% RSLogix 500 project P4_KOBIERSKI_M.RSS, saved by version 8.30.00.16 %
PROJECT "UNTITLED"    % processor: Bul.1763 MicroLogix 1100 Series B %

PROGRAM FILES
  LAD 2 "MAIN"  3 rungs
  LAD 3 "IO"  7 rungs
  LAD 4 "CYCLE"  11 rungs
  LAD 5 "STATES"  7 rungs

DATA FILES
  O0 OUTPUT  4 elements
  I1 INPUT  6 elements
  S2 STATUS  66 elements
  B3 BINARY  3 elements
  T4 TIMER  3 elements
  C5 COUNTER  1 elements
  R6 CONTROL  1 elements
  N7 INTEGER  2 elements
  F8 FLOAT  1 elements

LADDER 2 "MAIN"
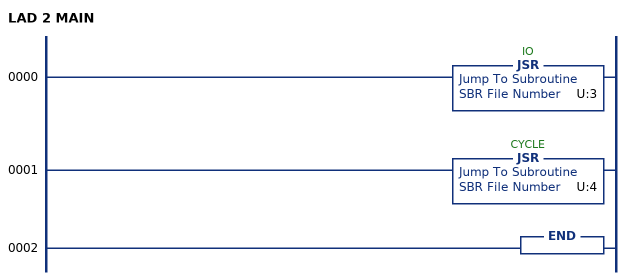
% Rung: 0 %
SOR JSR U:3 EOR
%   U:3  "IO" %
% Rung: 1 %
SOR JSR U:4 EOR
%   U:4  "CYCLE" %
% Rung: 2 %
SOR END EOR

LADDER 3 "IO"
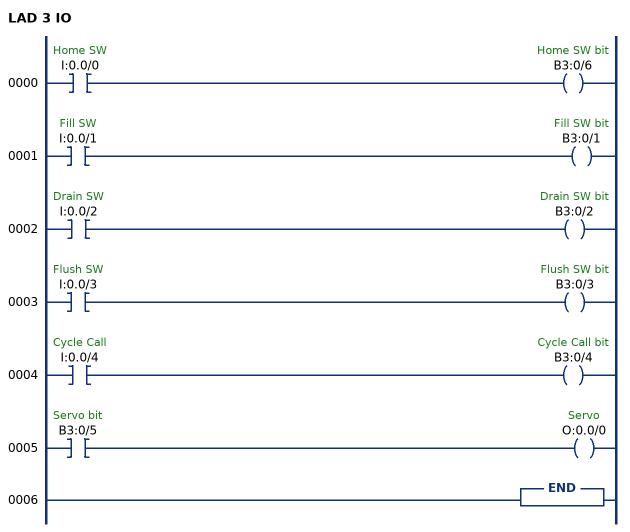
% Rung: 0 %
SOR XIC I:0.0/0 OTE B3:0/6 EOR
%   I:0.0/0  "Home SW" %
%   B3:0/6  "Home SW bit" %
% Rung: 1 %
SOR XIC I:0.0/1 OTE B3:0/1 EOR
%   I:0.0/1  "Fill SW" %
%   B3:0/1  "Fill SW bit" %
% Rung: 2 %
SOR XIC I:0.0/2 OTE B3:0/2 EOR
%   I:0.0/2  "Drain SW" %
%   B3:0/2  "Drain SW bit" %
% Rung: 3 %
SOR XIC I:0.0/3 OTE B3:0/3 EOR
%   I:0.0/3  "Flush SW" %
%   B3:0/3  "Flush SW bit" %
% Rung: 4 %
SOR XIC I:0.0/4 OTE B3:0/4 EOR
%   I:0.0/4  "Cycle Call" %
%   B3:0/4  "Cycle Call bit" %
% Rung: 5 %
SOR XIC B3:0/5 OTE O:0.0/0 EOR
%   B3:0/5  "Servo bit" %
%   O:0.0/0  "Servo" %
% Rung: 6 %
SOR END EOR

LADDER 4 "CYCLE"
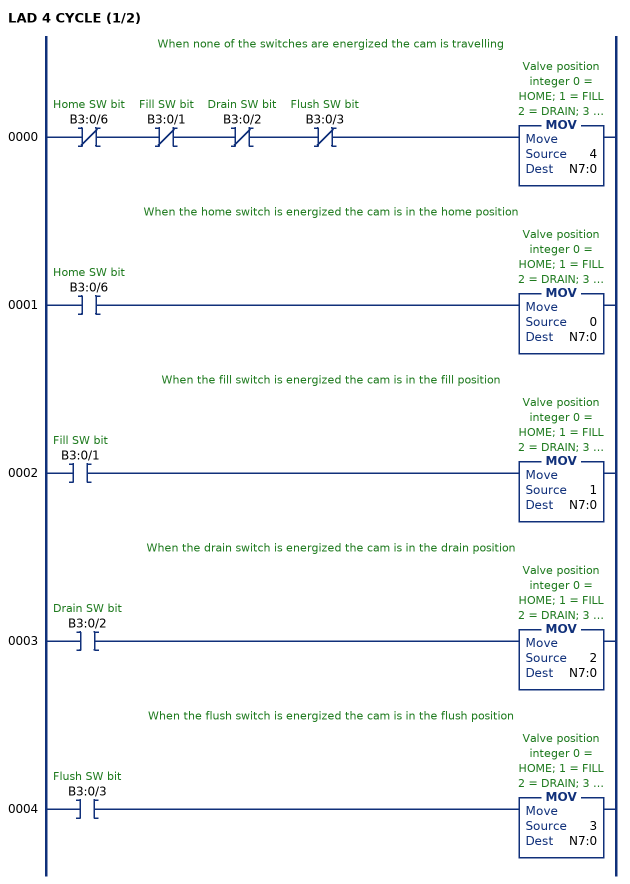
% Rung: 0 %
% When none of the switches are energized the cam is travelling %
SOR XIO B3:0/6 XIO B3:0/1 XIO B3:0/2 XIO B3:0/3 MOV 4 N7:0 EOR
%   B3:0/6  "Home SW bit" %
%   B3:0/1  "Fill SW bit" %
%   B3:0/2  "Drain SW bit" %
%   B3:0/3  "Flush SW bit" %
%   N7:0  "Valve position integer 0 = HOME; 1 = FILL 2 = DRAIN; 3 = FLUSH 4 = TRAVELLING" %
% Rung: 1 %
% When the home switch is energized the cam is in the home position %
SOR XIC B3:0/6 MOV 0 N7:0 EOR
%   B3:0/6  "Home SW bit" %
%   N7:0  "Valve position integer 0 = HOME; 1 = FILL 2 = DRAIN; 3 = FLUSH 4 = TRAVELLING" %
% Rung: 2 %
% When the fill switch is energized the cam is in the fill position %
SOR XIC B3:0/1 MOV 1 N7:0 EOR
%   B3:0/1  "Fill SW bit" %
%   N7:0  "Valve position integer 0 = HOME; 1 = FILL 2 = DRAIN; 3 = FLUSH 4 = TRAVELLING" %
% Rung: 3 %
% When the drain switch is energized the cam is in the drain position %
SOR XIC B3:0/2 MOV 2 N7:0 EOR
%   B3:0/2  "Drain SW bit" %
%   N7:0  "Valve position integer 0 = HOME; 1 = FILL 2 = DRAIN; 3 = FLUSH 4 = TRAVELLING" %
% Rung: 4 %
% When the flush switch is energized the cam is in the flush position %
SOR XIC B3:0/3 MOV 3 N7:0 EOR
%   B3:0/3  "Flush SW bit" %
%   N7:0  "Valve position integer 0 = HOME; 1 = FILL 2 = DRAIN; 3 = FLUSH 4 = TRAVELLING" %

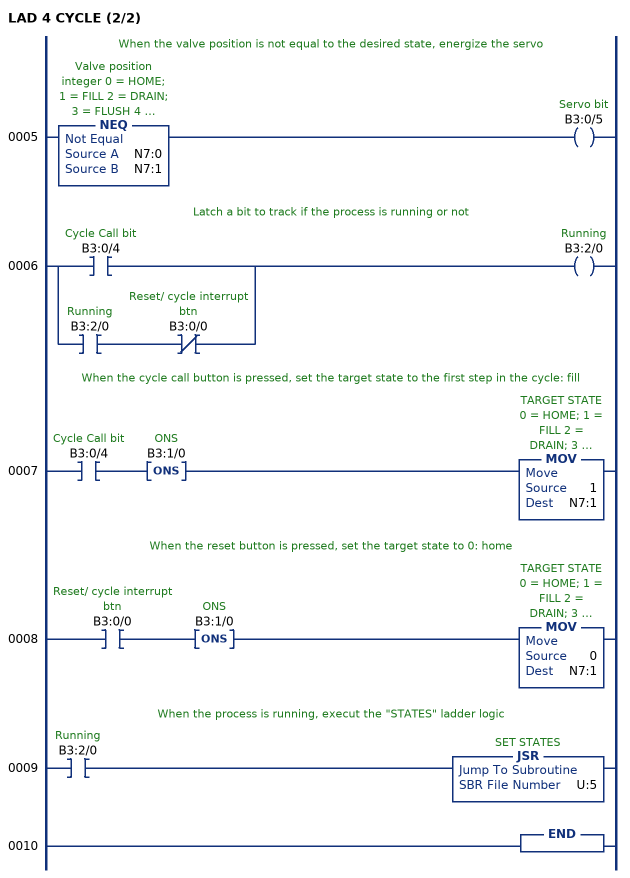
% Rung: 5 %
% When the valve position is not equal to the desired state, energize the servo %
SOR NEQ N7:0 N7:1 OTE B3:0/5 EOR
%   N7:0  "Valve position integer 0 = HOME; 1 = FILL 2 = DRAIN; 3 = FLUSH 4 = TRAVELLING" %
%   N7:1  "TARGET STATE 0 = HOME; 1 = FILL 2 = DRAIN; 3 = FLUSH" %
%   B3:0/5  "Servo bit" %
% Rung: 6 %
% Latch a bit to track if the process is running or not %
SOR BST XIC B3:0/4 NXB XIC B3:2/0 XIO B3:0/0 BND OTE B3:2/0 EOR
%   B3:0/4  "Cycle Call bit" %
%   B3:2/0  "Running" %
%   B3:0/0  "Reset/ cycle interrupt btn" %
% Rung: 7 %
% When the cycle call button is pressed, set the target state to the first step in the cycle: fill %
SOR XIC B3:0/4 ONS B3:1/0 MOV 1 N7:1 EOR
%   B3:0/4  "Cycle Call bit" %
%   B3:1/0  "ONS" %
%   N7:1  "TARGET STATE 0 = HOME; 1 = FILL 2 = DRAIN; 3 = FLUSH" %
% Rung: 8 %
% When the reset button is pressed, set the target state to 0: home %
SOR XIC B3:0/0 ONS B3:1/0 MOV 0 N7:1 EOR
%   B3:0/0  "Reset/ cycle interrupt btn" %
%   B3:1/0  "ONS" %
%   N7:1  "TARGET STATE 0 = HOME; 1 = FILL 2 = DRAIN; 3 = FLUSH" %
% Rung: 9 %
% When the process is running, execut the "STATES" ladder logic %
SOR XIC B3:2/0 JSR U:5 EOR
%   B3:2/0  "Running" %
%   U:5  "SET STATES" %
% Rung: 10 %
SOR END EOR

LADDER 5 "STATES"
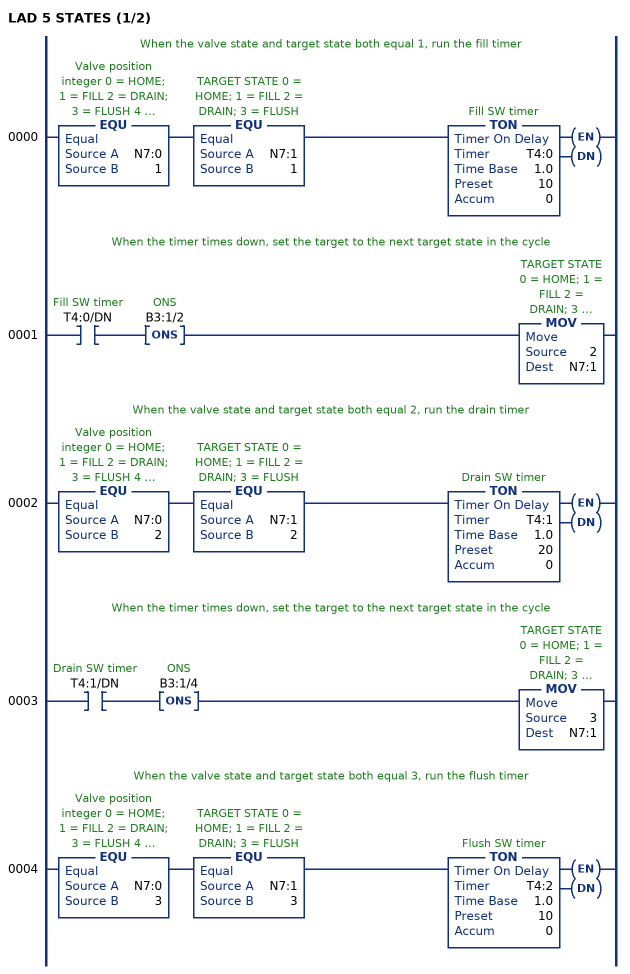
% Rung: 0 %
% When the valve state and target state both equal 1, run the fill timer %
SOR EQU N7:0 1 EQU N7:1 1 TON T4:0 1.0 10 0 EOR
%   N7:0  "Valve position integer 0 = HOME; 1 = FILL 2 = DRAIN; 3 = FLUSH 4 = TRAVELLING" %
%   N7:1  "TARGET STATE 0 = HOME; 1 = FILL 2 = DRAIN; 3 = FLUSH" %
%   T4:0  "Fill SW timer" %
% Rung: 1 %
% When the timer times down, set the target to the next target state in the cycle %
SOR XIC T4:0/DN ONS B3:1/2 MOV 2 N7:1 EOR
%   T4:0  "Fill SW timer" %
%   B3:1/2  "ONS" %
%   N7:1  "TARGET STATE 0 = HOME; 1 = FILL 2 = DRAIN; 3 = FLUSH" %
% Rung: 2 %
% When the valve state and target state both equal 2, run the drain timer %
SOR EQU N7:0 2 EQU N7:1 2 TON T4:1 1.0 20 0 EOR
%   N7:0  "Valve position integer 0 = HOME; 1 = FILL 2 = DRAIN; 3 = FLUSH 4 = TRAVELLING" %
%   N7:1  "TARGET STATE 0 = HOME; 1 = FILL 2 = DRAIN; 3 = FLUSH" %
%   T4:1  "Drain SW timer" %
% Rung: 3 %
% When the timer times down, set the target to the next target state in the cycle %
SOR XIC T4:1/DN ONS B3:1/4 MOV 3 N7:1 EOR
%   T4:1  "Drain SW timer" %
%   B3:1/4  "ONS" %
%   N7:1  "TARGET STATE 0 = HOME; 1 = FILL 2 = DRAIN; 3 = FLUSH" %
% Rung: 4 %
% When the valve state and target state both equal 3, run the flush timer %
SOR EQU N7:0 3 EQU N7:1 3 TON T4:2 1.0 10 0 EOR
%   N7:0  "Valve position integer 0 = HOME; 1 = FILL 2 = DRAIN; 3 = FLUSH 4 = TRAVELLING" %
%   N7:1  "TARGET STATE 0 = HOME; 1 = FILL 2 = DRAIN; 3 = FLUSH" %
%   T4:2  "Flush SW timer" %

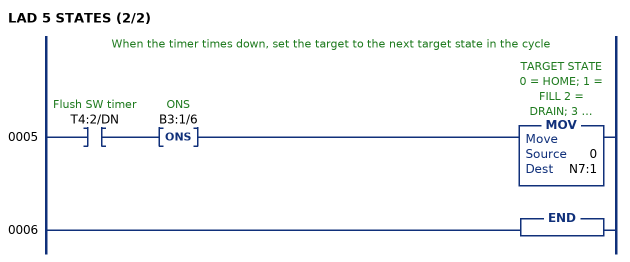
% Rung: 5 %
% When the timer times down, set the target to the next target state in the cycle %
SOR XIC T4:2/DN ONS B3:1/6 MOV 0 N7:1 EOR
%   T4:2  "Flush SW timer" %
%   B3:1/6  "ONS" %
%   N7:1  "TARGET STATE 0 = HOME; 1 = FILL 2 = DRAIN; 3 = FLUSH" %
% Rung: 6 %
SOR END EOR

OTHER DOCUMENTED ADDRESSES
  B3:0/7  "Reset/ Interrupt"
  B3:1/1  "ONS"
  B3:1/3  "ONS"
  B3:1/5  "ONS"

COMMENTS NOT ATTACHED TO A CURRENT RUNG
  N7:1: When the cycle call button is pressed, set the target state to the first step in the cycle: fill
  N7:0: When the drain switch is energized the cam is in the drain position

DATA TABLE (non-zero values as saved)
DATA T4
% .PRE .ACC %
% T4:0 % 10 0
% T4:1 % 20 0
% T4:2 % 10 0
